// TwinCAT 3 PLC project ProJsonBeckhoff
// Title: ProJsonBeckhoff
// Company: Michal Gasper
// Author: Michal Gasper
// ProjectVersion: 1.0.0.2
// Description: Fork from CODESYS library: https://forge.codesys.com/lib/pro-json/home/Home/
// ProgramVersion: 3.1.4026.19
// libraries:
//   Tc2_Standard, * (Beckhoff Automation GmbH)
//   Tc2_System, * (Beckhoff Automation GmbH)
//   Tc2_Utilities, * (Beckhoff Automation GmbH)
//   SysMem,3.5.17.0,System
// project tree:
//   Data Types/ ASCII.TcDUT, JSONNAMEVALUE.TcDUT, JSONVALUETYPE.TcDUT, JSONVAR.TcPOU, JSONVARNAME.TcDUT
//   Examples/ EXAMPLEJSONSTRUCT.TcDUT, EXAMPLEJSONSTRUCT_1.TcDUT, ExampleJSON_FB.TcPOU, ExampleJSON_PRG.TcPOU
//   Functions/ CLEANSTRING.TcPOU, ISBOOLEAN.TcPOU, ISNUMBER.TcPOU, JSON_TO_STRUCT.TcPOU, REAL_TO_STRING_X.TcPOU, SPLIT_VARNAME.TcPOU, STRUCT_TO_JSON.TcPOU
//   / GPL_JSON.TcGVL, Notes.TcPOU, PlcTask.TcTTO
// real-time tasks:
//   TASK PlcTask: cycle T#100000us, priority 20, ADS port 350

CONFIGURATION ProJsonBeckhoff
    RESOURCE PLC ON TwinCAT3
        TASK PlcTask(INTERVAL := T#100000us, PRIORITY := 20);
        PROGRAM MAIN WITH PlcTask : MAIN;
    END_RESOURCE
END_CONFIGURATION

// ---- Data Types/ASCII.TcDUT
TYPE ASCII :
(
	NULL := 0,
	SOH := 1,
	STX := 2,
	ETX := 3,
	EOT := 4,
	ENQ := 5,
	ACK := 6,
	BEL := 7,
	BS := 8,
	HT := 9,
	LF := 10,
	VT := 11,
	FF := 12,
	CR := 13,
	SO := 14,
	SI := 15,
	DLE := 16,
	DC1 := 17,
	DC2 := 18,
	DC3 := 19,
	DC4 := 20,
	NAK := 21,
	SYN := 22,
	ETB := 23,
	CAN := 24,
	EM := 25,
	SUB_ := 26,
	ESC := 27,
	FS := 28,
	GS := 29,
	RS := 30,
	US := 31,
	SPACE := 32,
	BANG := 33,
	DOUBLE_QUOTE := 34,
	HASH := 35,
	DOLLAR := 36,
	PERCENT := 37,
	AMPERSAND := 38,
	SINGLE_QUOTE := 39,
	OPEN_PAREN := 40,
	CLOSE_PAREN := 41,
	STAR := 42,
	PLUS := 43,
	COMMA := 44,
	MINUS := 45,
	DOT := 46,
	SLASH := 47,
	NUMBER_0 := 48,
	NUMBER_1 := 49,
	NUMBER_2 := 50,
	NUMBER_3 := 51,
	NUMBER_4 := 52,
	NUMBER_5 := 53,
	NUMBER_6 := 54,
	NUMBER_7 := 55,
	NUMBER_8 := 56,
	NUMBER_9 := 57,
	COLON := 58,
	SEMICOLON := 59,
	LESS_THAN := 60,
	EQUALS := 61,
	GREATER_THAN := 62,
	QUESTION := 63,
	AT_SIGN := 64,
	UPPERCASE_A := 65,
	UPPERCASE_B := 66,
	UPPERCASE_C := 67,
	UPPERCASE_D := 68,
	UPPERCASE_E := 69,
	UPPERCASE_F := 70,
	UPPERCASE_G := 71,
	UPPERCASE_H := 72,
	UPPERCASE_I := 73,
	UPPERCASE_J := 74,
	UPPERCASE_K := 75,
	UPPERCASE_L := 76,
	UPPERCASE_M := 77,
	UPPERCASE_N := 78,
	UPPERCASE_O := 79,
	UPPERCASE_P := 80,
	UPPERCASE_Q := 81,
	UPPERCASE_R := 82,
	UPPERCASE_S := 83,
	UPPERCASE_T := 84,
	UPPERCASE_U := 85,
	UPPERCASE_V := 86,
	UPPERCASE_W := 87,
	UPPERCASE_X := 88,
	UPPERCASE_Y := 89,
	UPPERCASE_Z := 90,
	OPEN_BRACKET := 91,
	BACKSLASH := 92,
	CLOSE_BRACKET := 93,
	CARET := 94,
	UNDERSCORE := 95,
	BACKQUOTE := 96,
	LOWERCASE_A := 97,
	LOWERCASE_B := 98,
	LOWERCASE_C := 99,
	LOWERCASE_D := 100,
	LOWERCASE_E := 101,
	LOWERCASE_F := 102,
	LOWERCASE_G := 103,
	LOWERCASE_H := 104,
	LOWERCASE_I := 105,
	LOWERCASE_J := 106,
	LOWERCASE_K := 107,
	LOWERCASE_L := 108,
	LOWERCASE_M := 109,
	LOWERCASE_N := 110,
	LOWERCASE_O := 111,
	LOWERCASE_P := 112,
	LOWERCASE_Q := 113,
	LOWERCASE_R := 114,
	LOWERCASE_S := 115,
	LOWERCASE_T := 116,
	LOWERCASE_U := 117,
	LOWERCASE_V := 118,
	LOWERCASE_W := 119,
	LOWERCASE_X := 120,
	LOWERCASE_Y := 121,
	LOWERCASE_Z := 122,
	OPEN_BRACE := 123,
	PIPE := 124,
	CLOSE_BRACE := 125,
	TILDE := 126,
	DEL := 127
) BYTE;
END_TYPE

// ---- Data Types/JSONNAMEVALUE.TcDUT
TYPE JSONNAMEVALUE :
STRUCT
	///name of the object at this level
	Name: STRING;
	///value of the object at this level
	Value: STRING;
	///array index of the object at this level
	ArrayIndex: UINT;
	IsArray: BOOL;
END_STRUCT
END_TYPE

// ---- Data Types/JSONVALUETYPE.TcDUT
TYPE JSONVALUETYPE :
(
	///local var is type STRING
	json_string,
	///local var is REAL
	json_number,
	///local var is DINT
	json_integer,
	///local var is BOOL
	json_boolean,
	///local var is type null
	json_null,
	///object is an array
	json_array,
	///object is another object (nested objects)
	json_object
);
END_TYPE

// ---- Data Types/JSONVARNAME.TcDUT
TYPE JSONVARNAME :
STRUCT
	///name of this variable or object
	Name: STRING(GPL_JSON.MAX_NAME_SIZE);
	///array index of the object at this level
	ArrayIndex: UINT;
	///first variable of a new object
	NewObject: BOOL;
	///last variable of an object
	EndObject: BOOL;
	///first variable of a new array
	NewArray: BOOL;
	///last variable of an array
	EndArray: BOOL;
END_STRUCT
END_TYPE

// ---- Examples/EXAMPLEJSONSTRUCT.TcDUT
TYPE EXAMPLEJSONSTRUCT :
STRUCT
	var1: JSONVAR;
	var2: JSONVAR;
	var3: JSONVAR;
	obj: EXAMPLEJSONSTRUCT_1;
	arrayobj: ARRAY[1..3] OF JSONVAR;
END_STRUCT
END_TYPE

// ---- Examples/EXAMPLEJSONSTRUCT_1.TcDUT
TYPE EXAMPLEJSONSTRUCT_1 :
STRUCT
	var4: JSONVAR;
	var5: JSONVAR;
	var6: JSONVAR;
	var7: ARRAY[1..3] OF JSONVAR;
END_STRUCT
END_TYPE

// ---- GPL_JSON.TcGVL
{attribute 'parameterlist' := ''}
{attribute 'qualified_only' := ''}
VAR_GLOBAL CONSTANT
	///maximum number of nested objects or array dimensions
	MAX_LEVELS: UINT := 10;
	///max string length of JSON name
	MAX_NAME_SIZE: UINT := 20;
	///max value string in bytes (all values are this size in memory)
	MAX_VALUE_SIZE: UINT := 50;
	///maximum length of full variable name with path
	MAX_VAR_NAME: UINT := 150;
	///maximum number of variables in the local structure
	MAX_VARS: UINT := 500;
	///maximum time for a single scan of the JSON_TO_STRUCT function block
	MAX_EXECUTION_TIME: TIME := TIME#50ms;
	///maximum allowable size of JSON string
	MAX_JSON_STRING: UINT := 20000;
	///formatting string for new line
	NEWLINE: STRING(2) := '$R$N';
	///formatting string for indentation
	INDENT: STRING(1) := '$T';
END_VAR

// ---- Functions/JSON_TO_STRUCT.TcPOU
FUNCTION_BLOCK JSON_TO_STRUCT
VAR_INPUT
	Execute:			BOOL;		//rising edge triggers parse of JSON string
	Abort:				BOOL;		//rising edge stops parsing of JSON string
	{attribute 'displaymode':='hex'}JSONString:		POINTER TO ARRAY[1..GPL_JSON.MAX_JSON_STRING] OF BYTE;	//pointer to JSON string
	JSONStringSize:		UDINT;		//size of string
	JSONVars:			POINTER TO ARRAY[1..GPL_JSON.MAX_VARS] OF JSONVAR;	//pointer to local structure made up of type JSONVAR
	NumberOfVars:		UINT;		//number of variables in the local structure or array
END_VAR

VAR_OUTPUT
	Busy:				BOOL;		//busy parsing a string
	Done:				BOOL;		//successfully parsed the whole string with no errors
	Aborted:			BOOL;		//parsing aborted by Abort input
	Error:				BOOL;		//unexpected character detected, string not completely parsed
	ErrorPosition:		UDINT;		//character position where the unexpected character was found
	ParseTime:			TIME;		//time it took to parse the string
END_VAR

VAR
	bufferposition:		UDINT;	//current position in the string
	NameValue:			ARRAY[1..GPL_JSON.MAX_LEVELS] OF JSONNAMEVALUE;	//name:value pairs currently being worked on
	obj_level:			UINT;	//number of nested objects
	name_start:			UDINT;	//index of the beginning of a name
	name_stop:			UDINT;	//index of the end of a name
	value_start:		UDINT;	//index of the beginning of a value
	value_stop:			UDINT;	//index of the end of a value
	findname:			BOOL;	//look for name in configuration array
	foundname:			BOOL;	//found a matching name in configuration array
	i:					UDINT;	//loop indexes
	jsonvarindex:		UINT;
	levelindex:			UINT;
	nameindex:			UINT;
	names:				ARRAY[1..GPL_JSON.MAX_LEVELS] OF JSONVARNAME;	//temp variable--can't access an array property
	thisloopstarttime:	TIME;		//time the current loop started
	starttime:			TIME;		//time parsing started
	Execute_TRIG:		R_TRIG;
	Abort_TRIG:			R_TRIG;
	findloop:			UINT;
	parse:				BOOL;
END_VAR

(*=======================================================================================================
JSON_TO_STRUCT()
Author: Tim Van Meppelen, Pro Electric Inc.
timv@proelectric.com
Date: Nov 2, 2018
parse JSON string and place the values in a matching local structure of type JSONVAR
========================================================================================================*)
thisloopstarttime:= TIME();	//store the time of the beginning of this loop	

Execute_TRIG(CLK:= Execute);
Abort_TRIG(CLK:= Abort);

IF Execute_TRIG.Q THEN
//must see a rising edge on execute to start parsing
	starttime:= TIME();	//store the time of the beginning of execution
	parse:= TRUE;
	bufferposition:= 1;
	Busy:= TRUE;
	Aborted:= FALSE;
	Done:= FALSE;
	Error:= FALSE;
	ErrorPosition:= 0;
	obj_level:= 0;
	FOR i:= 1 TO GPL_JSON.MAX_LEVELS DO
		NameValue[i].Name:= '';
		NameValue[i].Value:= '';
		NameValue[i].IsArray:= FALSE;
		NameValue[i].ArrayIndex:= 0;
	END_FOR
END_IF

IF Abort_TRIG.Q THEN
	Busy:= FALSE;
	Aborted:= TRUE;
	parse:= FALSE;
END_IF

(*====================PARSE JSON STRING====================*)
//parse the input string, and start storing values in NameValue array
WHILE parse DO
	IF (JSONString^[bufferposition] = ASCII.NULL) OR (bufferposition > JSONStringSize) THEN
	//strings are terminated with a null character
	//there might not always be a null character, for example in a network buffer that is stored as an array of bytes
		parse:= FALSE;
		Done:= TRUE;
		Busy:= FALSE;
		ParseTime:= TIME() - starttime;
		RETURN;
	END_IF	

	CASE JSONString^[bufferposition] OF 

	ASCII.DOUBLE_QUOTE:	// " name string
		Name();
		
	ASCII.OPEN_BRACE:// {, beginning of object
		OpenObject();	
		
	ASCII.CLOSE_BRACE:// }, end of object
		CloseObject();
		
	ASCII.OPEN_BRACKET:	// [, beginning of array
		OpenArray();
		
	ASCII.CLOSE_BRACKET:	// ], end of array
		CloseArray();
		
	ASCII.COLON:	// :, separator for name:value pairs
		Value();
		
	ASCII.COMMA:	// , move to next object
		Comma();
	
	ASCII.SOH..ASCII.SPACE:	// skip all control characters, including spaces
		bufferposition:= bufferposition + 1;

	ELSE
	//error, unexpected character
		ErrorHandler();
	END_CASE
	
	(*========================================LOOK FOR NAMES IN LOCAL VARIABLES========================================*)
	IF findname THEN
	//there is at least one valid name:value pair in the NameValue array--check for a match in the Config array, including nested objects
		findname:= FALSE;
		FOR findloop:= 1 TO NumberOfVars DO
		(*loop through all configured objects and look for the name that is currently being worked on in the JSON string
		Local JSON object should be as closely matched to the expected JSON string as possible, to decrease parsing speed.  
		This function will eventually find all objects, but it will start looking after the previous found variable, as it 
		is assumed that that's the most likely position for the next variable*)  
			jsonvarindex:= (jsonvarindex MOD NumberOfVars) + 1;
			names:= JSONVars^[jsonvarindex].Names;	//temporary variable
			FOR nameindex:= 1 TO obj_level DO
			//Match name and array index.  Array index will be 0 if the current name:value is not part of an array
				IF (names[nameindex].Name = NameValue[obj_level-(nameindex-1)].Name AND (NameValue[obj_level-(nameindex-1)].ArrayIndex = names[nameindex].ArrayIndex)) THEN	
					foundname:= TRUE;	//name in JSON string matches the local variable name
				ELSE
					foundname:= FALSE;	//name in JSON string does not match the local variable name, go to next name
					EXIT;
				END_IF
			END_FOR
			IF foundname THEN
				EXIT;
			END_IF
		END_FOR
	
		(*====================FOUND NAME, WRITE LOCAL VAR====================*)
		IF foundname THEN
		//local var name matches with JSON string name
			foundname:= FALSE;
			JSONVars^[jsonvarindex].AsString:= NameValue[obj_level].Value;	
		END_IF
	END_IF

	IF TIME() >= (thisloopstarttime + GPL_JSON.MAX_EXECUTION_TIME) THEN
	//this function block won't take up more than GPL_JSON.MAX_EXECUTION_TIME on one scan
	//very long strings or files could take too long to parse in one task cycle, and cause a watchdog exception
		RETURN;
	END_IF
END_WHILE

METHOD CloseArray
VAR_INPUT
END_VAR
(*=======================================================================================================
CloseArray()
end of an array
	
========================================================================================================*)

NameValue[obj_level].IsArray:= FALSE;
NameValue[obj_level].ArrayIndex:= 0;
bufferposition:= bufferposition + 1;
END_METHOD

METHOD CloseObject
VAR
	shiftindex:			INT;
END_VAR
(*=======================================================================================================
CloseObject()
end of an object, move down in the object hierarchy
========================================================================================================*)

NameValue[obj_level].Name:= '';
NameValue[obj_level].Value:= '';
NameValue[obj_level].IsArray:= FALSE;
NameValue[obj_level].ArrayIndex:= 0;
obj_level:= obj_level - 1;
bufferposition:= bufferposition + 1;
END_METHOD

METHOD Comma
VAR_INPUT
END_VAR
(*=======================================================================================================
Comma()
found a comma, parse an array value, or move on to the next object	
========================================================================================================*)

IF NameValue[obj_level].IsArray THEN
//if this is an array at the current object level, increment the array index
	NameValue[obj_level].ArrayIndex:= NameValue[obj_level].ArrayIndex + 1;
	Value();
ELSE
	bufferposition:= bufferposition + 1;
END_IF
END_METHOD

METHOD ErrorHandler
VAR_INPUT
END_VAR
(*=======================================================================================================
Error()
Unexpected or invalid character found, end parsing

========================================================================================================*)

parse:= FALSE;
Busy:= FALSE;
Error:= TRUE;
ErrorPosition:= bufferposition;	//return buffer position of unexpected character
RETURN;
END_METHOD

METHOD Name
VAR
	namestringok:		BOOL;
	j:					UDINT;
END_VAR
(*=======================================================================================================
Name()
found the first quote at the beginning of a name string,
extract the name string and put it into the NameValue array
========================================================================================================*)

name_start:= bufferposition + 1;
FOR j:= name_start TO (name_start+GPL_JSON.MAX_NAME_SIZE) DO
	IF (JSONString^[j] = 16#22) THEN
	//find the closing quote of a name string
		name_stop:= j - 1;		//name ends at character before quote
		bufferposition:= j + 1;	//next loop can start after the quote
		namestringok:= TRUE;
		EXIT;
	END_IF
END_FOR

IF namestringok THEN
	SysMemSet(
		pDest:= ADR(NameValue[obj_level].Name), 
		udiValue:= 0, 
		udiCount:= SIZEOF(NameValue[obj_level].Name)
	);
	
	SysMemCpy(
		pDest:= ADR(NameValue[obj_level].Name), 
		pSrc:= ADR(JSONString^[name_start]), 
		udiCount:= (name_stop+1 - name_start)
	);
ELSE
	ErrorHandler();
END_IF
END_METHOD

METHOD OpenArray
VAR_INPUT
END_VAR
(*=======================================================================================================
OpenArray()
found the beginning of an array, set array definition at this object level
========================================================================================================*)

NameValue[obj_level].IsArray:= TRUE;
NameValue[obj_level].ArrayIndex:= 1;
bufferposition:= bufferposition + 1;
END_METHOD

METHOD OpenObject
VAR
	shiftindex:			INT;
END_VAR
(*=======================================================================================================
OpenObject()
found the beginning of a new object, increment the object level
========================================================================================================*)

obj_level:= obj_level + 1;	//move up a level in the object hierarchy
bufferposition:= bufferposition + 1;
END_METHOD

METHOD Value
VAR
	valueloop:		UDINT;
	lookforname:	BOOL;
	j:				UDINT;
END_VAR
(*=======================================================================================================
Value()
found a ":" character, possible next characters are any combination of the following:
{ begin another object
[ begin a new array
" or a number or letter: value found
after all { and [ are found, and if any were found, the next thing will be a name string
loop through until a value is found, incrementing obj_level or array definitions as necessary
========================================================================================================*)

bufferposition:= bufferposition + 1;	//start searching after the ":" character
FOR valueloop:= 1 TO 20 DO 
//loop through the next 20 characters (maximum) looking for a value
	CASE JSONString^[bufferposition] OF
		
	ASCII.OPEN_BRACE:// {, beginning of new object
		OpenObject();	
		lookforname:= TRUE;
	
	ASCII.OPEN_BRACKET:	// [, beginning of new array
		OpenArray();
		
	ELSE
		IF lookforname THEN
		//a new object or array was found, and all nested objects have already been looped through, therefore this buffer position must start a new name
		//there is no value here, so exit this loop, main loop should now continue at the name, and parse its name:value pair
			EXIT;
		END_IF
		
		IF (JSONString^[bufferposition] = ASCII.DOUBLE_QUOTE) THEN
		//value starts with a quote character--quoted string
			value_start:= bufferposition + 1;	//value follows : and "	
		ELSE
			value_start:= bufferposition;	//value immediately follows :
		END_IF
		FOR j:= value_start TO (value_start+GPL_JSON.MAX_VALUE_SIZE) DO
			IF (JSONString^[j] = ASCII.DOUBLE_QUOTE)  THEN
			//end of value is is found at the closing quote
				value_stop:= j - 1;
				bufferposition:= j + 1;	//main loop can resume at the next character after the quote
				EXIT;
			ELSIF (JSONString^[j] = ASCII.COMMA) OR (JSONString^[j] = ASCII.CLOSE_BRACE) OR (JSONString^[j] = ASCII.CLOSE_BRACKET) THEN
			//end of value is is found at , or }, or ]
				value_stop:= j - 1;
				bufferposition:= j;	//main loop can resume at the next character after the value
				EXIT;
			END_IF
			IF (j = (value_start+GPL_JSON.MAX_VALUE_SIZE)) THEN
			//no closing quote was found after MAXVALUESIZE characters
				ErrorHandler();
			END_IF
		END_FOR	
		
		//clear previous string
		SysMemSet(
			pDest:= ADR(NameValue[obj_level].Value), 
			udiValue:= 0, 
			udiCount:= SIZEOF(NameValue[obj_level].Value)
		);
		//copy buffer to temporary value (string type)
		SysMemCpy(
			pDest:= ADR(NameValue[obj_level].Value), 
			pSrc:= ADR(JSONString^[value_start]), 
			udiCount:= (value_stop+1) - value_start 
		);	
		findname:= TRUE;		//there is a name:value pair in the NameValue array, check for a match with a local variable
		EXIT;
	END_CASE
END_FOR
END_METHOD

END_FUNCTION_BLOCK

// ---- Data Types/JSONVAR.TcPOU
{attribute 'pack_mode' := '4'}
{attribute 'reflection' := ''}
{attribute 'symbol' := 'none'}
FUNCTION_BLOCK JSONVAR
VAR_OUTPUT
	///properties can't be linked to visualizations, so this output var is updated every time AsString property is set
	{attribute 'symbol' := 'read'}
	HMIVarAsString: STRING(GPL_JSON.MAX_VALUE_SIZE);
END_VAR
VAR_STAT
	///highest variable name in previous variable
	{attribute 'hide'}
	PrevParentVar: REFERENCE TO INT;
	///path of the previous variable
	{attribute 'hide'}
	PrevNameArray: REFERENCE TO ARRAY [1..GPL_JSON.MAX_LEVELS] OF JSONVARNAME;
END_VAR
VAR
	///JSON name uses the variable name
	{attribute 'instance-path' := ''}
	{attribute 'noinit'}
	_VarNameFull: STRING(GPL_JSON.MAX_VAR_NAME);
	///variable path as an array. [1] is variable name, [2..x] are higher level structures
	_VarNameArray: ARRAY[1..GPL_JSON.MAX_LEVELS] OF JSONVARNAME;
	///type of variable contained in the value field, also implicity defines size of local var
	{attribute 'hide'}
	_ValueType: JSONVALUETYPE := JSONVALUETYPE.json_null;
	///value stored internally as an array of bytes
	{attribute 'hide'}
	_InternalValue: ARRAY[1..(GPL_JSON.MAX_VALUE_SIZE + 1)] OF BYTE;
	///size of internal value in bytes, automatically determined when any of the type properties are set
	{attribute 'hide'}
	_Size: UINT;
	///array position which points to the highest variable name
	{attribute 'hide'}
	_ParentVar: INT;
END_VAR

(*=======================================================================================================
JSONVAR()
Author: Tim Van Meppelen, Pro Electric Inc.
timv@proelectric.com
Date: Nov 2, 2018
local JSON variables

for use with JSON_TO_STRUCT, STRUCT_TO_JSON
variable type and size are automatically determined when a value is set, either:
	-with the set accessor of the AsString Property, which will make a guess at the type, based on the value
	-with any of the set accessors of the CharString, Boolean, Integer, Number, or Null properties
variable name is set automatically in FB_Init
	-variable name is the JSON name
	-JSON allows some object names that are not valid variable names in IEC61131, for example "type", 
	"3h", etc.  Workaround is to put an underscore at the beginning of the variable name.  This will
	match in JSON_TO_STRUCT, and STRUCT_TO_JSON will create a name without the leading underscore
========================================================================================================*)

{attribute 'monitoring' := 'call'}
PROPERTY AsString : STRING(GPL_JSON.MAX_VALUE_SIZE)
GET
(*=======================================================================================================
JSONVAR.AsString.Get()
Author: Tim Van Meppelen, Pro Electric Inc.
timv@proelectric.com
Date: Nov 2, 2018

get the variable value as a string
========================================================================================================*)

CASE _ValueType OF
JSONVALUETYPE.json_null:
	AsString:= 'null';
JSONVALUETYPE.json_boolean:
	IF THIS^.Boolean THEN
		AsString:= 'true';
	ELSE
		AsString:= 'false';
	END_IF
JSONVALUETYPE.json_number:
	AsString:= REAL_TO_STRING_X(THIS^.Number);
JSONVALUETYPE.json_integer:
	AsString:= DINT_TO_STRING(THIS^.Integer);
JSONVALUETYPE.json_string:
	AsString:= THIS^.CharString;
END_CASE
END_GET
SET
VAR
	TempBool: BOOL;
	TempReal: REAL;
	TempInt: DINT;
	TempString: STRING(255);
END_VAR
(*=======================================================================================================
JSONVAR.AsString.Set()
Author: Tim Van Meppelen, Pro Electric Inc.
timv@proelectric.com
Date: Nov 2, 2018

set the variable value as a string
========================================================================================================*)

IF (_ValueType = JSONVALUETYPE.json_null) THEN
//if the type is not explicitly configured, make a guess at the type
	IF ISNUMBER(ADR(AsString)) THEN
		_ValueType:= JSONVALUETYPE.json_number;
	ELSIF ISBOOLEAN(ADR(AsString)) THEN
		_ValueType:= JSONVALUETYPE.json_boolean;
	ELSIF (AsString = null) THEN
		_ValueType:= JSONVALUETYPE.json_null;
	ELSE
		_ValueType:= JSONVALUETYPE.json_string;
	END_IF
END_IF

CASE _ValueType OF
JSONVALUETYPE.json_null:
	THIS^.Null:= 'null';
JSONVALUETYPE.json_boolean:
	F_ToUCase(AsString);
	IF (AsString = 'TRUE') THEN
		TempBool:= TRUE;
	ELSE
		TempBool:= FALSE;
	END_IF
	THIS^.Boolean:= TempBool;
JSONVALUETYPE.json_number:
	TempReal:= STRING_TO_REAL(AsString);
	THIS^.Number:= TempReal;
JSONVALUETYPE.json_string:
	THIS^.CharString:= AsString;
END_CASE

HMIVarAsString:= AsString;
END_SET
END_PROPERTY

PROPERTY Boolean : BOOL
GET
(*=======================================================================================================
JSONVAR.Boolean.Get()
Author: Tim Van Meppelen, Pro Electric Inc.
timv@proelectric.com
Date: Nov 2, 2018

get a a boolean variable from the internal value
========================================================================================================*)

Boolean:= BYTE_TO_BOOL(_InternalValue[1]);
END_GET
SET
(*=======================================================================================================
JSONVAR.Boolean.set()
Author: Tim Van Meppelen, Pro Electric Inc.
timv@proelectric.com
Date: Nov 2, 2018

this is a boolean variable, copy to internal value and set type and size
========================================================================================================*)


_ValueType:= JSONVALUETYPE.json_boolean;
_Size:= 1;

//clear memory
SysMemSet(
	pDest:= ADR(_InternalValue), 
	udiValue:= 0, 
	udiCount:= SIZEOF(_InternalValue)
);

//put data into internal value
SysMemCpy(
	pDest:= ADR(_InternalValue), 
	pSrc:= ADR(Boolean), 
	udiCount:= _Size
);
END_SET
END_PROPERTY

PROPERTY CharString : STRING(GPL_JSON.MAX_VALUE_SIZE)
GET
VAR
	TempVar: STRING(255);
END_VAR
(*=======================================================================================================
JSONVAR.CharString.Get()
Author: Tim Van Meppelen, Pro Electric Inc.
timv@proelectric.com
Date: Nov 2, 2018

get a string variable from the internal value
========================================================================================================*)

SysMemCpy(
	pDest:= ADR(TempVar), 
	pSrc:= ADR(_InternalValue), 
	udiCount:= _Size+1
);
CharString:= TempVar;
END_GET
SET
(*=======================================================================================================
JSONVAR.CharString.Set()
Author: Tim Van Meppelen, Pro Electric Inc.
timv@proelectric.com
Date: Nov 2, 2018

this is a string variable, copy to internal value and set type and size
========================================================================================================*)

_ValueType:= JSONVALUETYPE.json_string;
_Size:= INT_TO_UINT(LEN(CharString));

//clear memory
SysMemSet(
	pDest:= ADR(_InternalValue), 
	udiValue:= 0, 
	udiCount:= SIZEOF(_InternalValue)
);

//put data into internal value
SysMemCpy(
	pDest:= ADR(_InternalValue), 
	pSrc:= ADR(CharString), 
	udiCount:= _Size+1
);
END_SET
END_PROPERTY

METHOD FB_Init : BOOL
VAR_INPUT
	/// TRUE: the retain variables are initialized (reset warm / reset cold)
	bInitRetains: BOOL;
	/// TRUE: the instance will be copied to the copy code afterward (online change)
	bInCopyCode: BOOL;
END_VAR
VAR
	ArrayPosition: UINT := GPL_JSON.MAX_LEVELS;
	NameStringPtr: POINTER TO ARRAY[1..GPL_JSON.MAX_VAR_NAME] OF BYTE;
	StringIndex: INT;
	VarNameBegin: INT;
	VarNameEnd: INT;
	VarNameIndex: INT;
	offset: INT;
	startarraystr: INT;
	endarraystr: INT;
	varlevelindex: INT;
	prevvarlevelindex: INT;
	stoploop: INT;
	startloop: INT;
END_VAR
(*=======================================================================================================
JSONVAR.FB_Init()
Author: Tim Van Meppelen, Pro Electric Inc.
timv@proelectric.com
Date: Nov 2, 2018
split the variable path into an array, and determine some object characteristics
example variable path: 'Test_M241.Test_M241.Application.TestJSON_PRG.TestStruct.var1'

TO DO:  objects and arrays should automatically close, as it is possible that this variable is the last one
the following variable should close an array or object through PrevNameArray

========================================================================================================*)

//====================GET VARIABLE NAME INTO AN ARRAY====================
NameStringPtr:= ADR(_VarNameFull);
StringIndex:= LEN(_VarNameFull);
VarNameEnd:= StringIndex;
VarNameIndex:= 1;

//TO DO:  use SPLIT function to create an array first, then loop through the array
WHILE (StringIndex > 0) DO
	IF (NameStringPtr^[StringIndex] = ASCII.DOT) THEN
		//found a "." character
		VarNameBegin:= StringIndex + 1;
		
		//clear array string  TO DO:  IS THIS NECESSARY?
		SysMemSet(
			pDest:= ADR(_VarNameArray[VarNameIndex]), 
			udiValue:= 0, 
			udiCount:= GPL_JSON.MAX_NAME_SIZE
		);

		//copy string between VarNameBegin and VarNameEnd
		SysMemCpy(
			pDest:= ADR(_VarNameArray[VarNameIndex]), 
			pSrc:= ADR(NameStringPtr^[VarNameBegin]), 
			udiCount:= INT_TO_UDINT((VarNameEnd - VarNameBegin)+1)
		);
		
		//remove leading _ from the name, if present
		IF FIND(STR1:= _VarNameArray[VarNameIndex].Name, STR2:= '_') = 1 THEN
			_VarNameArray[VarNameIndex].Name:= DELETE(STR:= _VarNameArray[VarNameIndex].Name, LEN:= 1, POS:= 1);
		END_IF
		
		//check if this is an array, if yes then remove the array index from the variable name
		startarraystr:= FIND(STR1:= _VarNameArray[VarNameIndex].Name, STR2:= '[');
		endarraystr:= FIND(STR1:= _VarNameArray[VarNameIndex].Name, STR2:= ']');
		IF (startarraystr <> 0) AND (endarraystr <> 0) THEN
			_VarNameArray[VarNameIndex].ArrayIndex:= STRING_TO_UINT(MID(
				STR:= _VarNameArray[VarNameIndex].Name, 
				LEN:= endarraystr-startarraystr-1, 
				POS:= startarraystr+1
			));
			_VarNameArray[VarNameIndex].Name:= DELETE(
				STR:= _VarNameArray[VarNameIndex].Name, 
				LEN:= endarraystr-startarraystr+1, 
				POS:= startarraystr
			);
		END_IF
		
        // ORIGINAL CODE LOOKED FOR 'Application' HERE.
        // Removed to allow the loop to parse the full path first.
	
		VarNameIndex:= VarNameIndex + 1;
		VarNameEnd:= VarNameBegin - 2;	//end of the next variable name is known, store for next loop
		StringIndex:= VarNameBegin - 2;
	ELSE
		StringIndex:= StringIndex - 1;
	END_IF
END_WHILE

// Top 2 levels of the path are Task/System and Program, which should be ignored.
// e.g. PlcTask.ExampleJSON_PRG.LocalJSONObj.var1
// _VarNameArray: [1]=var1, [2]=LocalJSONObj, [3]=ExampleJSON_PRG, [4]=PlcTask
// LocalJSONObj (index 2) needs to be the root.
// VarNameIndex is 4 here. 4 - 2 = 2.
IF _ParentVar = 0 THEN
    _ParentVar := VarNameIndex - 2;
    // Safety check: ParentVar must be at least 1
    IF _ParentVar < 1 THEN _ParentVar := 1; END_IF
END_IF

//====================JSON OBJECT CHARACTERISTICS====================
//figure out whether this variable is the first value of a new JSON object, or if the previous variable is the last value of a JSON object
IF __ISVALIDREF(PrevNameArray) THEN
//check for valid reference--will be invalid when FB_Init is run on the first instance of JSONVAR
	offset:= _ParentVar - PrevParentVar;	//check if the variable names have shifted up or down
	IF (offset < 0) THEN
	//objects shifted down
		stoploop:= PrevParentVar - 1;
		startloop:= 1;
	ELSE
	//no shift, or shift up
		stoploop:= _ParentVar - 1;
		startloop:= offset + 1;
	END_IF
	FOR varlevelindex:= startloop TO stoploop DO
		prevvarlevelindex:= varlevelindex - offset;
		IF (offset < 0) AND (varlevelindex = 1) THEN
		//if objects have shifted down, then i-offset will never point to PrevNameArray[1]
		//the previous variable might need an array closed
			IF (PrevNameArray[1].ArrayIndex > 0) THEN
			//end array
				PrevNameArray[1].EndArray:= TRUE;
			END_IF	
		END_IF
		
		IF ((varlevelindex-offset) > 1) AND ((_VarNameArray[varlevelindex].Name <> PrevNameArray[prevvarlevelindex].Name) OR (_VarNameArray[varlevelindex].ArrayIndex <> PrevNameArray[prevvarlevelindex].ArrayIndex)) THEN
		//end previous object
			PrevNameArray[prevvarlevelindex].EndObject:= TRUE;	//close previous object	
		END_IF	
		
		IF (PrevNameArray[prevvarlevelindex].ArrayIndex > 0) AND (_VarNameArray[varlevelindex].Name <> PrevNameArray[prevvarlevelindex].Name) THEN
		//end array
			PrevNameArray[prevvarlevelindex].EndArray:= TRUE;
		END_IF		
	
		IF (_VarNameArray[varlevelindex].ArrayIndex = 1) AND (PrevNameArray[prevvarlevelindex].ArrayIndex = 0) THEN
		//new array
			_VarNameArray[varlevelindex].NewArray:= TRUE;				
		END_IF	
	
		IF (varlevelindex > 1) AND ((NOT _VarNameArray[varlevelindex].NewArray) AND (_VarNameArray[varlevelindex].Name <> PrevNameArray[prevvarlevelindex].Name) OR (_VarNameArray[varlevelindex].ArrayIndex <> PrevNameArray[prevvarlevelindex].ArrayIndex)) THEN
		//new object
			_VarNameArray[varlevelindex].NewObject:= TRUE;	//new object at this level	
		END_IF	
	END_FOR

ELSE
//invalid reference to PrevNameArray, this must be the first variable
	FOR varlevelindex:= 1 TO _ParentVar-1 DO
		IF (varlevelindex > 1) THEN
		//every level above 1 will be a new object
			_VarNameArray[varlevelindex].NewObject:= TRUE;
		END_IF
		IF (_VarNameArray[varlevelindex].ArrayIndex = 1) THEN
		//new array
			_VarNameArray[varlevelindex].NewArray:= TRUE;				
		END_IF			
	END_FOR
END_IF

//set a reference to some variables for the next JSON variable
PrevNameArray REF= _VarNameArray;
PrevParentVar REF= _ParentVar;
END_METHOD

PROPERTY Integer : DINT
GET
VAR
	TempVar: REAL;
END_VAR
(*=======================================================================================================
JSONVAR.Integer.Get()
Author: Tim Van Meppelen, Pro Electric Inc.
timv@proelectric.com
Date: Nov 2, 2018

get an integer variable from the internal value
all number types are stored internally as floating point
========================================================================================================*)

SysMemCpy(
	pDest:= ADR(TempVar), 
	pSrc:= ADR(_InternalValue), 
	udiCount:= 4
);

Integer:= REAL_TO_DINT(TempVar);
END_GET
SET
VAR
	TempVar: REAL;
END_VAR
(*=======================================================================================================
JSONVAR.Integer.Set()
Author: Tim Van Meppelen, Pro Electric Inc.
timv@proelectric.com
Date: Nov 2, 2018

this is a integer variable, copy to internal value and set type and size
all number types are stored internally as floating point
========================================================================================================*)

_ValueType:= JSONVALUETYPE.json_integer;
_Size:= 4;

//clear memory
SysMemSet(
	pDest:= ADR(_InternalValue), 
	udiValue:= 0, 
	udiCount:= SIZEOF(_InternalValue)
);

TempVar:= DINT_TO_REAL(Integer);

//put data into internal value
SysMemCpy(
	pDest:= ADR(_InternalValue), 
	pSrc:= ADR(TempVar), 
	udiCount:= _Size
);
END_SET
END_PROPERTY

PROPERTY Names : ARRAY[1..GPL_JSON.MAX_LEVELS] OF JSONVARNAME
GET
Names:= _VarNameArray;
END_GET
END_PROPERTY

PROPERTY Null : STRING(4)
GET
(*=======================================================================================================
JSONVAR.Null.Get()
Author: Tim Van Meppelen, Pro Electric Inc.
timv@proelectric.com
Date: Nov 2, 2018

get a null value (returned as a string, as IEC61131 has no way to represent a null value)
========================================================================================================*)

Null:= 'null';
END_GET
SET
(*=======================================================================================================
JSONVAR.Null.Set()
Author: Tim Van Meppelen, Pro Electric Inc.
timv@proelectric.com
Date: Nov 2, 2018

this is a null variable, set type and size
========================================================================================================*)

_ValueType:= JSONVALUETYPE.json_null;
_Size:= 4;
END_SET
END_PROPERTY

PROPERTY Number : REAL
GET
VAR
	TempVar: REAL;
END_VAR
(*=======================================================================================================
JSONVAR.Number.Get()
Author: Tim Van Meppelen, Pro Electric Inc.
timv@proelectric.com
Date: Nov 2, 2018

get a floating point variable from the internal value
========================================================================================================*)

SysMemCpy(
	pDest:= ADR(TempVar), 
	pSrc:= ADR(_InternalValue), 
	udiCount:= 4
);
Number:= TempVar;
END_GET
SET
(*=======================================================================================================
JSONVAR.Number.Set()
Author: Tim Van Meppelen, Pro Electric Inc.
timv@proelectric.com
Date: Nov 2, 2018

this is a floating point variable, copy to internal value and set type and size
========================================================================================================*)

_ValueType:= JSONVALUETYPE.json_number;
_Size:= 4;

//clear memory
SysMemSet(
	pDest:= ADR(_InternalValue), 
	udiValue:= 0, 
	udiCount:= SIZEOF(_InternalValue)
);

//put data into internal value
SysMemCpy(
	pDest:= ADR(_InternalValue), 
	pSrc:= ADR(Number), 
	udiCount:= _Size
);
END_SET
END_PROPERTY

PROPERTY ParentVar : INT
GET
(*=======================================================================================================
JSONVAR.ParentVar.Get()
Author: Tim Van Meppelen, Pro Electric Inc.
timv@proelectric.com
Date: Nov 2, 2018

array position which points to the highest variable name
========================================================================================================*)

ParentVar:= _ParentVar;
END_GET
END_PROPERTY

{attribute 'monitoring' := 'call'}
PROPERTY Size : UINT
GET
(*=======================================================================================================
JSONVAR.Size.Get()
Author: Tim Van Meppelen, Pro Electric Inc.
timv@proelectric.com
Date: Nov 2, 2018

//size of internal value in bytes, automatically determined when any of the type properties are set
========================================================================================================*)

Size:= _Size;
END_GET
END_PROPERTY

{attribute 'monitoring' := 'call'}
PROPERTY ValueType : JSONVALUETYPE
GET
(*=======================================================================================================
JSONVAR.ValueType.Get()
Author: Tim Van Meppelen, Pro Electric Inc.
timv@proelectric.com
Date: Nov 2, 2018

type of variable contained in the value field, also implicity defines size of local var
========================================================================================================*)

ValueType:= _ValueType;
END_GET
END_PROPERTY

PROPERTY VarName : STRING(GPL_JSON.MAX_NAME_SIZE)
GET
(*=======================================================================================================
JSONVAR.VarName.Get()
Author: Tim Van Meppelen, Pro Electric Inc.
timv@proelectric.com
Date: Sept 16, 2019

get the name of the variable as a string, ie.
'Test_M241.Test_M241.Application.TestJSON_PRG.TestStruct.var1'

========================================================================================================*)

VarName:= _VarNameFull;
END_GET
SET
VAR
	Levels: UINT;
	i: INT;
END_VAR
(*=======================================================================================================
JSONVAR.SetVarName()
Author: Tim Van Meppelen, Pro Electric Inc.
timv@proelectric.com
Date: Sept 16, 2019

Manually set JSON variable name to something other than it's automatically generated name.  This should only 
be used when the JSON string could have a changing variable name at runtime, ie. the variable name is a date 
or a counter.  Normally, the JSON variable name is the same as the PLC variable name
NOTE:  this cannot change the number of levels of a nested object, it is assumed that the basic structure
remains the same, and only the names are changing

example created by FB_Init:
_VarNameFull   'Test_M241.Application.TestJSON_PRG.TestStruct.var1'
_VarNameArray                 [4]        [3]          [2]     [1]
_ParentVar = 2

example after runtime changes
_VarNameFull   'TestStruct.var1'
_VarNameArray      [2]     [1]
_ParentVar = 2

set as a string ie. 'TestStruct.var1'
each object inside another object must be changed manually
higher level object names must be changed in each lower level object
program level and above are not manually adjustable at runtime ie. 'Test_M241.Application.TestJSON_PRG.'

========================================================================================================*)

Levels:= SPLIT_VARNAME(VarNameArray:= _VarNameArray, StringIn:= VarName);

FOR i:= UINT_TO_INT(Levels) TO 1 BY -1 DO 
//recreate the var name string
	IF (i=UINT_TO_INT(Levels)) THEN
		_VarNameFull:= CONCAT(_VarNameArray[i].Name,'.');
	ELSIF (i=1) THEN
		_VarNameFull:= CONCAT(_VarNameFull, _VarNameArray[i].Name);
	ELSE
		_VarNameFull:= CONCAT(_VarNameFull, _VarNameArray[i].Name);
		_VarNameFull:= CONCAT(_VarNameFull, '.');
	END_IF
END_FOR
END_SET
END_PROPERTY

END_FUNCTION_BLOCK

// ---- Functions/REAL_TO_STRING_X.TcPOU
FUNCTION REAL_TO_STRING_X : STRING
VAR_INPUT
	In_REAL: REAL;
END_VAR
VAR
	TempVar: STRING;
END_VAR

(*=======================================================================================================
REAL_TO_STRING_X()
Author: Tim Van Meppelen, Pro Electric Inc.
timv@proelectric.com
Date: Nov 2, 2018
Standard REAL_TO_STRING function will always add a decimal place even if the input is a whole number
this function will drop the ".0" on the string output
========================================================================================================*)

TempVar:= REAL_TO_STRING(In_REAL);
IF (RIGHT(STR:= TempVar, SIZE:= 2) = '.0') THEN
	REAL_TO_STRING_X:= DELETE(STR:= TempVar, LEN:= 2, POS:= LEN(TempVar) - 1);
ELSE
	REAL_TO_STRING_X:= TempVar;
END_IF

END_FUNCTION

// ---- Functions/ISNUMBER.TcPOU
FUNCTION ISNUMBER : BOOL
VAR_INPUT
	In:		POINTER TO ARRAY[1..255] OF BYTE;
END_VAR
VAR
	i:				UINT;
	founddecimal:	BOOL;
END_VAR

(*=======================================================================================================
ISINTEGER()
Author: Tim Van Meppelen, Pro Electric Inc.
timv@proelectric.com
Date: Oct 2, 2018
check if a string contains a valid number, allows for "-" at the beginning of the string, and one "." character
========================================================================================================*)

FOR i:= 1 TO 256 DO
	CASE In^[i] OF 	
	ASCII.NULL:
	//end of string
		EXIT;
	ASCII.MINUS:
	//only allow a "-" in the first position	
		IF (i=1) THEN
			ISNUMBER:= TRUE;
		ELSE
			ISNUMBER:= FALSE;
			EXIT;
		END_IF
	ASCII.DOT:
	//only allow one decimal point
		IF founddecimal THEN
		//already found one decimal, can't have two
			ISNUMBER:= FALSE;
			EXIT;
		ELSE
		//first decimal point found, allow one
			ISNUMBER:= TRUE;
			founddecimal:= TRUE;
		END_IF
	ASCII.NUMBER_0..ASCII.NUMBER_9:
		ISNUMBER:= TRUE;
	ELSE
	//all other characters are not part of numbers
		ISNUMBER:= FALSE;
		EXIT;
	END_CASE
END_FOR

END_FUNCTION

// ---- Functions/ISBOOLEAN.TcPOU
FUNCTION ISBOOLEAN : BOOL
VAR_INPUT
	In:		POINTER TO STRING(5);
END_VAR
VAR
	TempVar:	STRING(5);
END_VAR

(*=======================================================================================================
ISBOOLEAN()
Author: Tim Van Meppelen, Pro Electric Inc.
timv@proelectric.com
Date: Oct 2, 2018
check if a string would convert to a valid boolean variable
========================================================================================================*)
TempVar:= In^;
F_ToUCase(TempVar);

ISBOOLEAN:= (TempVar = 'TRUE') OR (TempVar = 'FALSE');

END_FUNCTION

// ---- Functions/SPLIT_VARNAME.TcPOU
FUNCTION SPLIT_VARNAME : UINT
VAR_INPUT
	VarNameArray: REFERENCE TO ARRAY [1..GPL_JSON.MAX_LEVELS] OF JSONVARNAME;
	///input string
	StringIn: STRING(GPL_JSON.MAX_VAR_NAME);
END_VAR
VAR CONSTANT
	SPLIT_CHAR: STRING(1) := '.';
END_VAR
VAR
	ArraySize: UINT := 1;
	sShortString: STRING;
	iSplitLocation: INT;
	i: UINT;
	TempArray: ARRAY[1..GPL_JSON.MAX_LEVELS] OF STRING;
END_VAR

(*=======================================================================================================
SPLIT_VARNAME()
Author: Tim Van Meppelen, Pro Electric Inc.
timv@proelectric.com
Date: June 26, 2018
split a string into an array at the '.' character

TO DO:
'a.b.c.d' becomes an array[1]=d, [2]=c, [3]=b, [4]=a
modified from https://forum.codesys.com/viewtopic.php?t=9889
========================================================================================================*)

//Loop through string until there is no string left or array has hit its limits
WHILE (LEN(StringIn) > 0) DO
    //Find location of first break point
    iSplitLocation := FIND(STR1:= StringIn, STR2:= SPLIT_CHAR) - 1;

    //If there is no break point found then set location to size of string
    IF (iSplitLocation = -1) THEN 
        iSplitLocation := LEN(StringIn);
    END_IF
  
    //Copy the part of the string that is needed for the parameter.
    sShortString := MID(STR:= StringIn, LEN:= iSplitLocation, POS:= 1);

    //Make sure string is not empty before using up an array spot.
    IF (LEN(sShortString) > 0) THEN
        TempArray[ArraySize] := sShortString;
        ArraySize := ArraySize + 1;
    END_IF

    //Remove copied components from long string
    StringIn := DELETE(STR:= StringIn, LEN:= (iSplitLocation + 1), POS:= 1);

    //Check to see if more parameters can fit in array. If not exit loop
    IF (ArraySize > GPL_JSON.MAX_LEVELS) THEN
        EXIT;
    END_IF 
END_WHILE

ArraySize:= ArraySize - 1;

FOR i:= 0 TO ArraySize DO
    //Reverse the order of the array
    VarNameArray[i+1].Name:= TempArray[ArraySize-i];
END_FOR

SPLIT_VARNAME:= ArraySize;

END_FUNCTION

// ---- Examples/ExampleJSON_FB.TcPOU
FUNCTION_BLOCK ExampleJSON_FB
VAR
	LocalJSONObj: EXAMPLEJSONSTRUCT;
	ComposeJSON: STRUCT_TO_JSON;
	JSONString: STRING(1000);
	NewJSONObj: EXAMPLEJSONSTRUCT;
	ParseJSON: JSON_TO_STRUCT;
END_VAR

(*=======================================================================================================
ExampleJSON_FB()
example function block testing nested objects

========================================================================================================*)

LocalJSONObj.var1.Boolean:= TRUE;
LocalJSONObj.var2.Number:= 34.8756;
LocalJSONObj.var3.CharString:= 'teststring';
LocalJSONObj.obj.var4.Number:= 22;
LocalJSONObj.obj.var5.AsString:= 'FALSE';	//JSONVAR will guess at type, in this case, boolean
LocalJSONObj.obj.var6.CharString:= 'qwer';
LocalJSONObj.obj.var7[1].Number:= 123.234;
LocalJSONObj.obj.var7[2].AsString:= '55.46';	//JSONVAR will guess at type, in this case, a number
LocalJSONObj.obj.var7[3].Number:= 985;
LocalJSONObj.arrayobj[1].Number:= 1;
LocalJSONObj.arrayobj[2].Number:= 2;
LocalJSONObj.arrayobj[3].Number:= 3;

//create a JSON string from local object
ComposeJSON(
	JSONString:= ADR(JSONString), 
	JSONStringSize:= SIZEOF(JSONString),
	JSONVars:= ADR(LocalJSONObj),
	NumberOfVars:= SIZEOF(LocalJSONObj) / SIZEOF(JSONVAR)
);

//fill another local object with values from the created JSON string
ParseJSON(
	Execute:= ComposeJSON.Done,
	JSONString:= ADR(JSONString), 
	JSONStringSize:= SIZEOF(JSONString),
	JSONVars:= ADR(NewJSONObj),
	NumberOfVars:= SIZEOF(NewJSONObj) / SIZEOF(JSONVAR)
);

END_FUNCTION_BLOCK

// ---- Functions/STRUCT_TO_JSON.TcPOU
FUNCTION_BLOCK STRUCT_TO_JSON
VAR_INPUT
	Execute:			BOOL;		//rising edge triggers compose of JSON string
	Abort:				BOOL;		//rising edge stops composing a JSON string
	{attribute 'displaymode':='hex'}JSONString:		POINTER TO ARRAY[1..GPL_JSON.MAX_JSON_STRING] OF BYTE;	//pointer to JSON string
	JSONStringSize:		UDINT;		//size of string
	JSONVars:			POINTER TO ARRAY[1..GPL_JSON.MAX_VARS] OF JSONVAR;	//pointer to local structure made up of type JSONVAR
	NumberOfVars:		UINT;		//number of variables in the local structure or array
	VariableArraySize:	BOOL;		//don't write array values which are null, resulting in variable array sizes
	Format:				BOOL;		//add white space and indenting to the resulting string
END_VAR

VAR_OUTPUT
	Busy:				BOOL;		//busy composing a string
	Done:				BOOL;		//successfully composed the whole string with no errors
	Aborted:			BOOL;		//compose aborted by Abort input
	Error:				BOOL;		//unexpected character detected, string not completely composed
	ErrorPosition:		UDINT;		//index of local object at which composing stopped
	ComposeTime:		TIME;		//time it took to compose the string
END_VAR

VAR
	bufferposition:		UDINT;	//current position in the string
	jsonvarindex:		UDINT;
	compose:			BOOL;	
	objectstr:			STRING(255);	//string created by current variable
	names:				ARRAY[1..GPL_JSON.MAX_LEVELS] OF JSONVARNAME;	//helper variable for names array property
	namesindex:			INT;
	i:					UINT;
	
	Execute_TRIG:		R_TRIG;
	Abort_TRIG:			R_TRIG;
	thisloopstarttime:	TIME;		//time the current loop started
	starttime:			TIME;		//time composing started
END_VAR

(*=======================================================================================================
STRUCT_TO_JSON()
Author: Tim Van Meppelen, Pro Electric Inc.
timv@proelectric.com
Date: Nov 2, 2018
create a JSON string from a structure of JSONVAR types
========================================================================================================*)

thisloopstarttime:= TIME();	//store the time of the beginning of this loop

Execute_TRIG(CLK:= Execute);
Abort_TRIG(CLK:= Abort);

IF Execute_TRIG.Q THEN
//must see a rising edge on execute to start composing
	starttime:= TIME();	//store the time of the beginning of execution
	compose:= TRUE;
	Busy:= TRUE;
	Aborted:= FALSE;
	Done:= FALSE;
	Error:= FALSE;
	ErrorPosition:= 0;
	bufferposition:= 1;
	jsonvarindex:= 1;	
	FOR i:= 1 TO GPL_JSON.MAX_LEVELS DO
	//clear names array
		names[i].Name:= '';
		names[i].ArrayIndex:= 0;
	END_FOR
	//clear previous string
	SysMemSet(
		pDest:= JSONString, 
		udiValue:= 0, 
		udiCount:= JSONStringSize
	);
END_IF

IF Abort_TRIG.Q THEN
	Busy:= FALSE;
	Aborted:= TRUE;
	compose:= FALSE;
END_IF



WHILE compose AND (jsonvarindex <= NumberOfVars) AND (bufferposition < JSONStringSize) DO 
//loop through all local variables
	objectstr:= '';	//clear previous object string	
	names:= JSONVars^[jsonvarindex].Names;	//helper variable for name array property
	
	IF (jsonvarindex = 1) THEN
		objectstr:= CONCAT(objectstr, '{');	//open JSON string with {
		IF Format THEN
			objectstr:= CONCAT(objectstr, GPL_JSON.NEWLINE);
		END_IF
	ELSE
		IF NOT (VariableArraySize AND (names[1].ArrayIndex > 0) AND (JSONVars^[jsonvarindex].ValueType = JSONVALUETYPE.json_null)) THEN
		//don't write the value if the current variable is an array, and the value is null
			objectstr:= CONCAT(objectstr, ',');	//comma in between each value
			IF Format AND (names[1].ArrayIndex <= 1) THEN
			//new line after each comma, except in arrays
				objectstr:= CONCAT(objectstr, GPL_JSON.NEWLINE);	
			END_IF	
		END_IF

	END_IF

	FOR namesindex:= JSONVars^[jsonvarindex].ParentVar-1 TO 1 BY -1 DO 
	//start at the second highest variable level and count down
	//open new objects or arrays, and write a single name:value pair at level 1
		//======================open new objects or arrays, or create new name:value pairs======================
		IF names[namesindex].NewArray AND (names[namesindex].ArrayIndex <= 1) THEN
		//new array at this level
			CreateName(Name:= names[namesindex].Name);
			CreateArray();	
		END_IF	

		IF (jsonvarindex <> 1) AND (namesindex > 1) AND names[namesindex].NewObject THEN
		//new object at this level, don't create objects at level 1
			IF (names[namesindex].ArrayIndex = 0) THEN
			//only create an object name if this is not part of an array
				CreateName(Name:= names[namesindex].Name);
			END_IF
			CreateObject();	
		END_IF
		
		IF (namesindex=1) THEN
		//only write a value at level 1
			IF (names[namesindex].ArrayIndex > 0) THEN
			//array, create value only
				IF NOT (VariableArraySize AND (names[1].ArrayIndex > 0) AND (JSONVars^[jsonvarindex].ValueType = JSONVALUETYPE.json_null)) THEN
				//don't write the value if the current variable is an array, and the value is null
					CreateValue(ValueType:= JSONVars^[jsonvarindex].ValueType, Value:= JSONVars^[jsonvarindex].AsString);					
				END_IF
			ELSE
			//name:value pair
				CreateName(Name:= names[namesindex].Name);
				CreateValue(ValueType:= JSONVars^[jsonvarindex].ValueType, Value:= JSONVars^[jsonvarindex].AsString);
			END_IF
		END_IF
	END_FOR
	
	FOR namesindex:= 1 TO JSONVars^[jsonvarindex].ParentVar-1 DO 
	//start at the lowest level and count up
	//close objects or arrays if this is the last value in this object or array
		IF names[namesindex].EndObject THEN
		//close object at this level, unless it's the last object in the
			CloseObject();
		END_IF

		IF names[namesindex].EndArray THEN	
		//close array at this level
			CloseArray();	
		END_IF	
	END_FOR	
	
	//concatenate the temporary object string to the JSON string output
	SysMemCpy(
		pDest := ADR(JSONString^[bufferposition]),
		pSrc := ADR(objectstr),
		udiCount := INT_TO_UDINT(LEN(objectstr))
	);
	
	bufferposition:= bufferposition + DINT_TO_UDINT(LEN(objectstr));

	IF (jsonvarindex >= NumberOfVars) THEN
	//end of vars, close string
		compose:= FALSE;
		Busy:= FALSE;
		Done:= TRUE;		
		ComposeTime:= TIME() - starttime;
		//JSONString^[bufferposition]:= ASCII.CLOSE_BRACE;;	//close JSON object with }
		JSONString^[bufferposition]:= ASCII.NULL;	//null character to end string
	END_IF
	
	IF TIME() >= (thisloopstarttime + GPL_JSON.MAX_EXECUTION_TIME) THEN
	//this function block won't take up more than GPL_JSON.MAX_EXECUTION_TIME on one scan
	//very long strings could take too long to compose in one task cycle, and cause a watchdog exception
		RETURN;
	END_IF
	
	jsonvarindex:= jsonvarindex + 1;	
END_WHILE

METHOD CloseArray
VAR_INPUT
END_VAR
(*=======================================================================================================
CloseArray()
Author: Tim Van Meppelen, Pro Electric Inc.
timv@proelectric.com
Date: Oct 22, 2018
close a JSON array
========================================================================================================*)
objectstr:= CONCAT(objectstr, ']');

IF Format THEN
	objectstr:= CONCAT(objectstr, GPL_JSON.NEWLINE);	
END_IF
END_METHOD

METHOD CloseObject
VAR
	indent:		INT;
END_VAR
(*=======================================================================================================
CloseObject()
Author: Tim Van Meppelen, Pro Electric Inc.
timv@proelectric.com
Date: Oct 22, 2018
close a JSON object
========================================================================================================*)
IF Format THEN
	FOR indent:= 1 TO JSONVars^[jsonvarindex].ParentVar-1 DO
		objectstr:= CONCAT(objectstr, GPL_JSON.INDENT);	
	END_FOR
END_IF

objectstr:= CONCAT(objectstr, '}');
END_METHOD

METHOD CreateArray
VAR_INPUT
END_VAR
(*=======================================================================================================
CreateArray()
Author: Tim Van Meppelen, Pro Electric Inc.
timv@proelectric.com
Date: Oct 22, 2018
create a new JSON array

[ ------ ------------ value ---------------- ] 
        /                               \
	    \_______________ , _____________/
		
========================================================================================================*)
objectstr:= CONCAT(objectstr, '[');	//opening [
END_METHOD

METHOD CreateName
VAR_INPUT
	Name:	STRING(GPL_JSON.MAX_NAME_SIZE);
END_VAR
VAR
	indent:		INT;
END_VAR
(*=======================================================================================================
CreateName()
Author: Tim Van Meppelen, Pro Electric Inc.
timv@proelectric.com
Date: Oct 22, 2018
create a JSON name string from a local variable of type JSONVAR
========================================================================================================*)
IF Format THEN
	FOR indent:= 1 TO JSONVars^[jsonvarindex].ParentVar-1 DO
		objectstr:= CONCAT(objectstr, GPL_JSON.INDENT);	
	END_FOR
END_IF

objectstr:= CONCAT(objectstr, '"');	//opening quote
objectstr:= CONCAT(objectstr, Name);//variable name
objectstr:= CONCAT(objectstr, '":');	//closing quote and name:value separator
END_METHOD

METHOD CreateObject
VAR_INPUT
END_VAR
(*=======================================================================================================
CreateObject()
Author: Tim Van Meppelen, Pro Electric Inc.
timv@proelectric.com
Date: Oct 22, 2018
create a new JSON object

{------ "name" ------ : ----- value --------- }
        /                                 \
	    \_______________ , _______________/

========================================================================================================*)
objectstr:= CONCAT(objectstr, '{');	//opening {

IF Format THEN
	objectstr:= CONCAT(objectstr, GPL_JSON.NEWLINE);
END_IF
END_METHOD

METHOD CreateValue
VAR_INPUT
	ValueType:		JSONVALUETYPE;
	Value:			STRING(GPL_JSON.MAX_VALUE_SIZE);
END_VAR
(*=======================================================================================================
CreateValue()
Author: Tim Van Meppelen, Pro Electric Inc.
timv@proelectric.com
Date: Oct 22, 2018
create a JSON value string from a local variable of type JSONVAR
========================================================================================================*)
CASE ValueType OF
//append value to object string
JSONVALUETYPE.json_number:
	objectstr:= CONCAT(objectstr, Value);
JSONVALUETYPE.json_integer:
	objectstr:= CONCAT(objectstr, Value);	
JSONVALUETYPE.json_boolean:
	objectstr:= CONCAT(objectstr, Value);
JSONVALUETYPE.json_string:
	objectstr:= CONCAT(objectstr, '"');	//opening quote
	objectstr:= CONCAT(objectstr, Value);
	objectstr:= CONCAT(objectstr, '"');	//closing quote
JSONVALUETYPE.json_null:
	objectstr:= CONCAT(objectstr, 'null');
END_CASE
END_METHOD

METHOD ErrorHandler
VAR_INPUT
END_VAR
(*=======================================================================================================
Error()
Something went wrong, return the index of the variable where the problem was encountered
========================================================================================================*)

compose:= FALSE;
Busy:= FALSE;
Error:= TRUE;
ErrorPosition:= jsonvarindex;	//return buffer position of unexpected character
RETURN;
END_METHOD

END_FUNCTION_BLOCK

// ---- Examples/ExampleJSON_PRG.TcPOU
PROGRAM ExampleJSON_PRG
VAR
	LocalJSONObj: EXAMPLEJSONSTRUCT;
	ComposeJSON: STRUCT_TO_JSON;
	JSONString: STRING(1000);
	NewJSONObj: EXAMPLEJSONSTRUCT;
	ParseJSON: JSON_TO_STRUCT;
	
	ExampleJSON : ExampleJSON_FB;
END_VAR

(*=======================================================================================================
ExampleJSON_PRG()
Author: Tim Van Meppelen, Pro Electric Inc.
timv@proelectric.com
Date: Nov 2, 2018
example program demonstrating JSONVAR, STRUCT_TO_JSON, AND JSON_TO_STRUCT

This example will populate a structure with values and types.  On a rising edge of ComposeJSON.Execute, 
ComposeJSON will create a JSON string.  When ComposeJSON.Done is set, ParseJSON.Execute is set, and 
ParseJSON will parse that string back into a different structure.

Tested with 200mS cyclic task, GPL_JSON.MAX_EXECUTION_TIME=50mS
Depending on the application and speed of the controller, these values could be changed. 
Be aware of how much cycle time is being taken when using multiple function blocks.
Each function block will limit its time to GPL_JSON.MAX_EXECUTION_TIME, but multiple function blocks 
could take up more than that.  This is on the list of things that could be improved. 

JSONVAR
FB_Init will fill in information about the variable name and structure in VarNameArray
variable type and size are automatically determined when a value is set, either:
	-with the set accessor of the AsString Property, which will make a guess at the type, based on the value
	-with any of the set accessors of the CharString, Boolean, Integer, Number, or Null properties
variable name is set automatically in FB_Init
	-variable name is the JSON name
	-JSON allows some object names that are not valid variable names in IEC61131, for example "type", 
	"3h", etc.  Workaround is to put an underscore at the beginning of the variable name.  This will
	match in JSON_TO_STRUCT, and STRUCT_TO_JSON will create a name without the leading underscore
	
JSON_TO_STRUCT
convert a JSON string into a local structure of JSONVAR
Long strings can take several seconds--for example, I have tested with a string of 20kB length, and the 
parse time is about 4 seconds.  Ensuring that the local variable structure is designed to be as close as 
possible to the expected order of variables in the JSON string will decrease parsing time, the search loop 
always starts with the next local variable and loops around until a match is found.

STRUCT_TO_JSON
convert a local structure of JSONVAR to a JSON string
.Format input will create indenting and new lines, useful for writing to a file

GPL_JSON
Parameter list that contains limits on size of strings, arrays, etc.  Most of these variables are simply
to limit memory usage, so they can be increased or decreased to suit the local application and controller

========================================================================================================*)

LocalJSONObj.var1.Boolean:= TRUE;
LocalJSONObj.var2.Number:= 34.8756;
LocalJSONObj.var3.CharString:= 'teststring';
LocalJSONObj.obj.var4.Number:= 22;
LocalJSONObj.obj.var5.AsString:= 'FALSE';	//JSONVAR will guess at type, in this case, boolean
LocalJSONObj.obj.var6.CharString:= 'qwer';
LocalJSONObj.obj.var7[1].Number:= 123.234;
LocalJSONObj.obj.var7[2].AsString:= '55.46';	//JSONVAR will guess at type, in this case, a number
LocalJSONObj.obj.var7[3].Number:= 985;
LocalJSONObj.arrayobj[1].Number:= 1;
LocalJSONObj.arrayobj[2].Number:= 2;
LocalJSONObj.arrayobj[3].Number:= 3;

//create a JSON string from local object
ComposeJSON(
	JSONString:= ADR(JSONString), 
	JSONStringSize:= SIZEOF(JSONString),
	JSONVars:= ADR(LocalJSONObj),
	NumberOfVars:= SIZEOF(LocalJSONObj) / SIZEOF(JSONVAR)
);

//fill another local object with values from the created JSON string
ParseJSON(
	Execute:= ComposeJSON.Done,
	JSONString:= ADR(JSONString), 
	JSONStringSize:= SIZEOF(JSONString),
	JSONVars:= ADR(NewJSONObj),
	NumberOfVars:= SIZEOF(NewJSONObj) / SIZEOF(JSONVAR)
);

ExampleJSON();

END_PROGRAM

// ---- Functions/CLEANSTRING.TcPOU
FUNCTION CLEANSTRING : BOOL
VAR_INPUT
	StringPtr:		POINTER TO ARRAY[1..MAXSTRINGLENGTH] OF BYTE;
END_VAR
VAR CONSTANT
	MAXSTRINGLENGTH:	UINT:= 2048;
END_VAR
VAR
	i:				UINT;
	j:				UINT;
END_VAR

(*=======================================================================================================
CLEANSTRING()
Author: Tim Van Meppelen, Pro Electric Inc.
timv@proelectric.com
Date: Oct 9, 2018
strip all control characters and spaces from a string
========================================================================================================*)

FOR i:= 1 TO MAXSTRINGLENGTH DO
	IF (StringPtr^[i] >= 1) AND (StringPtr^[i] <= 16#20) THEN
	//match all control and white space characters, except for null, which terminates a string
		FOR j:= i TO MAXSTRINGLENGTH DO
			IF (StringPtr^[j] = 16#00) THEN
			//null character terminates string
				EXIT;
			ELSE
			//shift character array left one
				StringPtr^[j]:= StringPtr^[j+1];
			END_IF
		END_FOR
		i:= i - 1;	//run loop at same position again
	ELSIF (StringPtr^[i] = 16#00) THEN
	//found null character at the end of the string
		EXIT;
	END_IF
END_FOR

CLEANSTRING:= TRUE;

END_FUNCTION

// ---- Notes.TcPOU
PROGRAM Notes

(*=======================================================================================================
Notes
Author: Tim Van Meppelen, Pro Electric Inc.
timv@proelectric.com
current version 1.0.0.2
Last updated: March 6, 2019

BUGS
-STRUCT_TO_JSON/JSONVAR.FB_Init()
	-doesn't add the closing ] if it's the last item in the structure
	-doesn't add the closing } if a nested object is the last item in the structure
	-both of the above for the same reason--closing objects is done by the following object, see JSONVAR.FB_Init() line 70-115
	-what about setting EndObject to TRUE by default, and having the following object set it to FALSE if not a new object?
-all arrays must be 1 based, haven't investigated further with 0 based arrays
-STRUCT_TO_JSON 
	-Format input is partially implemented, needs more testing with various different strings and structures
	-should use spaces for indentation rather than tabs?
-JSON_TO_STRUCT.Value()
	-line 36: what happens if a value string is longer than MAX_VALUE_SIZE?

	
	
NEW IDEAS
-STRUCT_TO_JSON	
	-create variable length arrays on the JSON side if values are null?
-speed up
-JSON_STRINGIFY function that can be called multiple times to create a JSON string from key and value string inputs
	-would create JSON on the fly without having to define a JSONVAR structure
	-could be useful for small strings, HTTP server responses, etc
-Schneider SoMachine does not support the __NEW operator, but eventually this would be a better way to implement JSON_TO_STRUCT


VERSION HISTORY
-should start making better notes on version history








========================================================================================================*)

END_PROGRAM
